TYPE U_TIMESTRUCT :
UNION
	TIMESTRUCT : TIMESTRUCT;
	nWORD : ARRAY[1..8] OF WORD;
END_UNION
END_TYPE

(* stored: Version 1.1.0.1, ProductVersion 3.1.4024.12
   DUT U_TIMESTRUCT: Id {d3570536-eb24-428e-9741-c13176c5b680} *)
